{attribute 'GeneratedUsingTerminal: EL3443-0000-0016'}
{attribute addProperty BoxType "EL3443-0000-0016"}
{attribute addProperty Id "Voltage_Last_Zero_CrossingAT %I*ULINT8"}
{attribute addProperty CRC "3439292703"}
{attribute addProperty Size "8"}
TYPE L2_Timing_CCFF711F EXTENDS InputBase_8311D824 :
STRUCT
	{attribute addProperty Name "Voltage_Last_Zero_Crossing"}
	Voltage_Last_Zero_Crossing AT %I* : ULINT;
END_STRUCT
END_TYPE

(* stored: Version 1.2.0.0, ProductVersion 3.1.4024.9
   DUT L2_Timing_CCFF711F: Id {ec81a52e-9270-40d3-b954-2e5ea2ef8737} *)
